FUNCTION_BLOCK InfluentFeed (* CAT Function Block Type *)
  (* Standard: 61499-2 *)
  (* Version 0.0, 6/13/2026, Schneider Electric, template *)
  PACKAGE SE.Nereda;
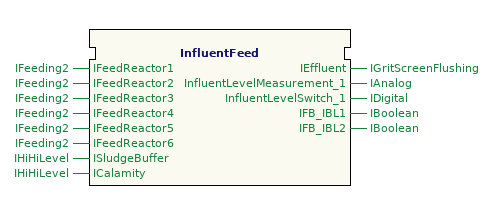
  SOCKETS
    IFeedReactor1 : IFeeding2;
    IFeedReactor2 : IFeeding2;
    IFeedReactor3 : IFeeding2;
    IFeedReactor4 : IFeeding2;
    IFeedReactor5 : IFeeding2;
    IFeedReactor6 : IFeeding2;
    ISludgeBuffer : IHiHiLevel;
    ICalamity : IHiHiLevel;
  END_SOCKETS
  PLUGS
    IEffluent : IGritScreenFlushing;
    InfluentLevelMeasurement_1 : IAnalog;
    InfluentLevelSwitch_1 : IDigital;
    IFB_IBL1 : IBoolean;
    IFB_IBL2 : IBoolean;
  END_PLUGS
  (* 01 - FUNCTIONNAL INPUT INTERFACE *)
  (* 00 - INITIALIZATION *)
  (* 05 - LOGIC *)
  (* 06 - HMI INTERFACE *)
  (* 02 - FUNCTIONNAL OUTPUT INTERFACE *)
  (* Influent Feed Logic *)
  (* 04 - CHILDREN *)
  (* 4A - TYPICALS *)
  (* Created by Nouriddin OUECHEN *)
  (* 03 - FIELD INTERFACE *)
  (* 07- REACTOR ALARM *)
  FBS
    INIT : plcStart(Prio := 50, Delay := T#0ms);
    IThis : InfluentFeed_HMI(QI := TRUE);
    Actuators : InfluentActuators;
    Sensors : InfluentSensors;
    InfluentFeedLogic : InfluentFeedLogic;
    CheckInfluentFeedPipe : ALARM_BIT(ACKTYPE_1 := 2, ACTIVE := TRUE, TYPE := 1);
    LevelTooHighInfluentBuffer : ALARM_BIT(ACKTYPE_1 := 2, ACTIVE := TRUE, TYPE := 1);
  END_FBS
  EVENT_CONNECTIONS
    INIT.FIRST_INIT TO IThis.4C2FD2FF19635CC3;
    INIT.REDO_INIT TO IThis.4C2FD2FF19635CC3;
    Sensors.257CDF5EC36D9721 TO InfluentFeedLogic.BC06CE1931362B8B;
    InfluentFeedLogic.F42AAFD6672A0845 TO CheckInfluentFeedPipe.INIT;
    IThis.0762D69A46409181 TO Actuators.CFECDF36D4CD32D8;
    Actuators.7DD79654DC794726 TO Sensors.9977DC17201CA619;
    CheckInfluentFeedPipe.CNF_INITDATA TO CheckInfluentFeedPipe.REQ;
    CheckInfluentFeedPipe.CNF_INITDATA TO CheckInfluentFeedPipe.ACTIVATE;
    LevelTooHighInfluentBuffer.INITO TO CheckInfluentFeedPipe.REQ_INITDATA;
    LevelTooHighInfluentBuffer.INITO TO INIT.ACK_FIRST;
    LevelTooHighInfluentBuffer.CNF_INITDATA TO LevelTooHighInfluentBuffer.ACTIVATE;
    LevelTooHighInfluentBuffer.CNF_INITDATA TO LevelTooHighInfluentBuffer.REQ;
    CheckInfluentFeedPipe.INITO TO LevelTooHighInfluentBuffer.INIT;
    LevelTooHighInfluentBuffer.INITO TO LevelTooHighInfluentBuffer.REQ_INITDATA;
    Sensors.409CEAF28252E4B1 TO LevelTooHighInfluentBuffer.REQ;
  END_CONNECTIONS
  DATA_CONNECTIONS
    Sensors.45B83F9CD0834A04 TO LevelTooHighInfluentBuffer.INP;
  END_CONNECTIONS
  ADAPTER_CONNECTIONS
    Sensors.2E67B850256E4773 TO InfluentFeedLogic.E1C86A9341152426;
    Sensors.E2A5BC3A235FB2EF TO InfluentFeedLogic.041EF78E075C55E1;
    Sensors.78391E2D4F46EFA1 TO InfluentFeedLogic.C214550B8DC42EF6;
    Sensors.40C65F09E8D61204 TO InfluentFeedLogic.016F8FD2526F89A7;
    Sensors.699D75E9FF6E8CE7 TO InfluentFeedLogic.01317810F3C73242;
    Sensors.B410C1B56735CF55 TO InfluentFeedLogic.79F70E44EB9C9F70;
    Sensors.CB8A2840F5C7AAC3 TO InfluentFeedLogic.0CAF03FE242F99E5;
    IFeedReactor1 TO InfluentFeedLogic.609F02705A399057;
    IFeedReactor2 TO InfluentFeedLogic.1F7AAC7B5106D4B2;
    IFeedReactor3 TO InfluentFeedLogic.7443219931057EA2;
    IFeedReactor4 TO InfluentFeedLogic.E9AC4665A13CBE6F;
    IFeedReactor5 TO InfluentFeedLogic.53E97B5155727226;
    IFeedReactor6 TO InfluentFeedLogic.5E0EC60B9A0D6B28;
    ISludgeBuffer TO InfluentFeedLogic.FD2779514DE73082;
    ICalamity TO InfluentFeedLogic.0A5A50004CB895CC;
    Sensors.F09DC5AC3C279647 TO InfluentFeedLogic.0527B216F6436059;
    Sensors.F209125E681BDB46 TO InfluentFeedLogic.6DF51F6AD72EB612;
    Actuators.0437085E1A4A1F82 TO InfluentFeedLogic.E7D1F137E38EA84F;
    InfluentFeedLogic.AD72937293C08D51 TO IEffluent;
    InfluentFeedLogic.4AFCD4E2D6EF6FC7 TO Actuators.4AEDE0FD7FB6C66C;
    InfluentFeedLogic.878EAB56847311CF TO Actuators.1E97C2475591089E;
    InfluentFeedLogic.2A2153EE89B36415 TO Actuators.980568D1DFD4B2B2;
    InfluentFeedLogic.0C7F28210482186E TO Actuators.6395F0AB68CF1389;
    InfluentFeedLogic.41A77D46AD024567 TO Actuators.FD732CD7A58EBF2B;
    InfluentFeedLogic.6A43EA2E48BEB575 TO Actuators.D247FD058B4CE88E;
    InfluentFeedLogic.AD9E2C7325E87035 TO Actuators.066706720A080036;
    InfluentFeedLogic.CA4F1A9DF212B4F7 TO Actuators.DAAD5510446F66AA;
    Sensors.55BCDD699EAC3442 TO InfluentFeedLogic.B7B2CCE4E357E20D;
    Sensors.17FB584A3AFD1EEC TO InfluentFeedLogic.14226A285C625124;
    Sensors.656137DBE41C10E7 TO InfluentFeedLogic.51607D0D1E29BF18;
    InfluentFeedLogic.B34E51ADAF028396 TO Actuators.0832F0F59B656E80;
    InfluentFeedLogic.67B29A684061473C TO Actuators.1816FE45B75B3650;
    Sensors.5C582A915C8D98D8 TO InfluentLevelMeasurement_1;
    Sensors.E8428DDA357DC0C4 TO InfluentLevelSwitch_1;
    Sensors.EB7B6D3A8E8E83E7 TO IFB_IBL1;
    Sensors.AFAD5E4DC964C45D TO IFB_IBL2;
  END_CONNECTIONS
END_FUNCTION_BLOCK
